INTERFACE ITF_ControlElement_HMI

METHOD LinkControlElementData : BOOL
VAR_INPUT
	stData				: REFERENCE TO ST_ControlElement_HMI_Link;
END_VAR
END_METHOD

END_INTERFACE

(* stored: Version 1.1.0.1, ProductVersion 3.1.4024.15
   Itf ITF_ControlElement_HMI: Id {9ab225a5-6d3a-489a-8f21-bf97c3be3e87}
   Method LinkControlElementData: Id {6809e73f-35c9-4469-9ccd-79e6c59c7c58} *)
